FUNCTION_BLOCK ABSTRACT FBA_Drive IMPLEMENTS I_Drive
VAR_INPUT
	bEnable : BOOL;
	//when a traverse sensor is opposite of this value, the respective property becomes TRUE
	//all sensors for a drive should be of the same type - do not mix & match PNP and NPN sensors on the same drive
END_VAR
(*
this abstract FB only specifies the minimum data for any drive
*)

{attribute 'monitoring':='call'}
PROPERTY ABSTRACT Active : BOOL
GET
END_GET
END_PROPERTY

{attribute 'monitoring':='call'}
PROPERTY ABSTRACT Error : BOOL
GET
END_GET
END_PROPERTY

{attribute 'TcRpcEnable'}
METHOD ABSTRACT reset : BOOL
VAR_INPUT
END_VAR
END_METHOD

{attribute 'TcRpcEnable'}
METHOD ABSTRACT stop : BOOL
VAR_INPUT
END_VAR
END_METHOD

END_FUNCTION_BLOCK

(* stored: Version 1.1.0.1, ProductVersion 3.1.4024.11
   POU FBA_Drive: Id {2de1cb23-32f2-4219-89c5-fb81e366fa09}, SpecialFunc None
   Folder Abstract: Id {c5aa1f87-afe2-4e7f-ace1-de8c3966dd88}
   Property Active: Id {d1381e43-e73a-47e2-a25c-0a860678c4a2}
   Get Get: Id {5e5510a3-652b-4cb8-aa27-d7e65ef261f6}
   Property Error: Id {f91f2d47-7f8e-4d3d-9a9c-df891ddd96e0}
   Get Get: Id {cf5a7583-df79-4b7c-9e12-e919740dc30d}
   Method reset: Id {89936125-0d83-4e3e-88d4-6abae24e37b7}
   Method stop: Id {b225f2f1-2348-4f1a-aec3-8bf30e5b2053} *)
